INTERFACE I_PersistentEventStorage

METHOD StoreEvent 
VAR_INPUT
	stEvent:ST_Event;
END_VAR
END_METHOD

END_INTERFACE

(* stored: Version 1.1.0.1, ProductVersion 3.1.4024.6
   Itf I_PersistentEventStorage: Id {38c59b76-86ea-414e-abb6-08135566f1a8}
   Method StoreEvent: Id {93648daf-c0e1-469a-b8b5-922b3efa53b5} *)
